FUNCTION_BLOCK PAEActDiverter EXTENDS PAEActuator2way_In
VAR_INPUT
END_VAR
VAR_OUTPUT
END_VAR
VAR
END_VAR

METHOD PUBLIC PAEActDiverter
VAR_INPUT
END_VAR
END_METHOD

END_FUNCTION_BLOCK

(* stored: Version 1.1.0.1, ProductVersion 3.1.4020.12
   POU PAEActDiverter: Id {e69dc658-0ccb-4ee7-b5c2-3b9ef93e7d53}, SpecialFunc None
   Method PAEActDiverter: Id {094f4704-69e6-4122-90d7-4b6e5d9586ea} *)
